# EPICS substitutions: iocBoot/iocCygwin/softMotor.substitutions
file "$(STD)/stdApp/Db/softMotor.db"
{
pattern
{P,		SM}
{xxx:,	SM1}
{xxx:,	SM2}
{xxx:,	SM3}
{xxx:,	SM4}
{xxx:,	SM5}
{xxx:,	SM6}
{xxx:,	SM7}
{xxx:,	SM8}
{xxx:,	SM9}
{xxx:,	SM10}
}
